// TIA Portal V19 export
DATA_BLOCK "TIMER DATA BLOCK"   // DB31
{ S7_Optimized_Access := 'TRUE' }
VERSION : 0.0
// stored: AutoNumber false, MemoryReserve 0
   VAR RETAIN
      COUNT_DOWN_TIMER_VALUE : S5Time;   // ACTUAL TIMER VALUE COUNT DOWN
      TIMER_SETP_ACTUAL_TIMER : S5Time;   // TIMER SETPOINT ACTUAL TIMER
      D_2 : S5Time;
      D_3 : S5Time;
      D_4 : S5Time;
      D_5 : S5Time;
      D_6 : S5Time;
      D_7 : S5Time;
      D_8 : S5Time;
      D_9 : S5Time;
      SETPOINT_TIMER_10 : S5Time;   // SETP.T10
      SETPOINT_TIMER_11 : S5Time;   // SETP.T11
      SETPOINT_TIMER_12 : S5Time;   // SETP.T12
      SETPOINT_TIMER_13 : S5Time;   // SETP.T13
      SETPOINT_TIMER_14 : S5Time := S5T#30M;   // SETP.T14 STERILE TIME
      SETPOINT_TIMER_15 : S5Time := S5T#10M;   // SETP.T15 COOLING TIME
      SETPOINT_TIMER_16 : S5Time := S5T#30S;   // SETP.T16 BLOW OUT CONDENSATE
      SETPOINT_TIMER_17 : S5Time := S5T#3M_20S;   // SETP.T17 BLOW OUT AFTER STOP
      SETPOINT_TIMER_18 : S5Time := S5T#3S;   // SETP.T18 DELAY OPEN 01.12
      SETPOINT_TIMER_19 : S5Time;   // SETP.T19
      SETPOINT_TIMER_20 : S5Time;   // SETP.T20
      SETPOINT_TIMER_21 : S5Time;   // SETP.T21
      SETPOINT_TIMER_22 : S5Time;   // SETP.T22
      SETPOINT_TIMER_23 : S5Time;   // SETP.T23
      SETPOINT_TIMER_24 : S5Time;   // SETP.T24
      SETPOINT_TIMER_25 : S5Time;   // SETP.T25
      SETPOINT_TIMER_26 : S5Time;   // SETP.T26
      SETPOINT_TIMER_27 : S5Time := S5T#4M;   // SETP.T27 PRERINSE
      SETPOINT_TIMER_28 : S5Time := S5T#2M_30S;   // SETP.T28 DOSING LYE
      SETPOINT_TIMER_29 : S5Time := S5T#30M;   // SETP.T29 CIRCULATION LYE
      SETPOINT_TIMER_30 : S5Time := S5T#10M;   // SETP.T30 INTERMEDIATE RINSE
      SETPOINT_TIMER_31 : S5Time := S5T#2M_20S;   // SETP.T31 DOSING ACID
      SETPOINT_TIMER_32 : S5Time := S5T#20M;   // SETP.T32 CIRCULATION ACID
      SETPOINT_TIMER_33 : S5Time := S5T#20M;   // SETP.T33 FINAL RINSE
      SETPOINT_TIMER_34 : S5Time := S5T#5M;   // SETP.T34 BLOW OUT AFTER CIP
      SETPOINT_TIMER_35 : S5Time := S5T#5S;   // SETP.T35 DELAY ALARM FILLING PRESSURE
      SETPOINT_TIMER_36 : S5Time := S5T#25S;   // SETP.T36 DELAY TT 01.76 BARRIER
      SETPOINT_TIMER_37 : S5Time := S5T#25S;   // SETP.T37 DELAY TT 01.78 BARRIER
      SETPOINT_TIMER_38 : S5Time := S5T#10S;   // SETP.T38 PAUSE TIME AGITATOR
      SETPOINT_TIMER_39 : S5Time := S5T#10S;   // SETP.T39 RUN TIME AGITATOR
      SETPOINT_TIMER_40 : S5Time := S5T#4S;   // SETP.T40 DELAY RESET STOP LIGHT
      SETPOINT_TIMER_41 : S5Time := S5T#10S;   // SETP.T41 DELAY ALARM STEAM
      SETPOINT_TIMER_42 : S5Time := S5T#10S;   // SETP.T42 DELAY ALARM AIR
      SETPOINT_TIMER_43 : S5Time := S5T#10S;   // SETP.T43 DELAY ALARM WATER
      SETPOINT_TIMER_44 : S5Time := S5T#5M;   // SETP.T44 DELAY BEFORE PURGING
      SETPOINT_TIMER_45 : S5Time := S5T#25S;   // SETP.T45 PURGING FILLING LINE
      SETPOINT_TIMER_46 : S5Time := S5T#2M;   // SETP.T46 PAUSE 01.13 PRESTE.
      SETPOINT_TIMER_47 : S5Time := S5T#1S;   // SETP.T47 OPEN 01.13 PRESTE.
      SETPOINT_TIMER_48 : S5Time := S5T#10S;   // SETP.T48 OPEN 01.13 CIP
      SETPOINT_TIMER_49 : S5Time := S5T#10S;   // SETP.T49 OPEN 01.18 CIP
      SETPOINT_TIMER_50 : S5Time := S5T#5S;   // SETP.T50 OPEN 01.24 CIP
      SETPOINT_TIMER_51 : S5Time := S5T#2M;   // SETP.T51 PAUSE BEFORE 01.08 OPEN
      SETPOINT_TIMER_52 : S5Time := S5T#5S;   // SETP.T52 FLIP 01.44 AT STOP FILLING
      SETPOINT_TIMER_53 : S5Time := S5T#15S;   // SETP.T53 DETERGENT CONC OK
      SETPOINT_TIMER_54 : S5Time := S5T#4M;   // SETP.T54 LYE DOSING TOO LONG
      SETPOINT_TIMER_55 : S5Time := S5T#4M;   // SETP.T55 ACID DOSING TOO LONG
      SETPOINT_TIMER_56 : S5Time := S5T#5S;   // SETP.T56
      SETPOINT_TIMER_57 : S5Time;   // SETP.T57
      SETPOINT_TIMER_58 : S5Time;   // SETP.T58
      SETPOINT_TIMER_59 : S5Time := S5T#5S;   // SETP.T59
      SETPOINT_TIMER_60 : S5Time := S5T#3S;   // SETP.T60
      D_61 : S5Time := S5T#3S;
      D_62 : S5Time;
      D_63 : S5Time;
      D_64 : S5Time;
      D_65 : S5Time;
      D_66 : S5Time;
      D_67 : S5Time;
      D_68 : S5Time;
      D_69 : S5Time;
      D_70 : S5Time;
   END_VAR
BEGIN
END_DATA_BLOCK
